# EPICS autosave request: CARSApp/Db/CARS_4_motor_positions.req
# FILE... CARS_8_CARS_motor_positions.req
file "CARS_motor_positions.req", P=$(P), M=m1
file "CARS_motor_positions.req", P=$(P), M=m2
file "CARS_motor_positions.req", P=$(P), M=m3
file "CARS_motor_positions.req", P=$(P), M=m4
